// TIA Portal V20 export
FUNCTION_BLOCK "Tippler"   // FB400, LAD
{ S7_Optimized_Access := 'TRUE' }
// stored: AutoNumber false, MemoryReserve 100, SetENOAutomatically false
   VAR_INPUT
      Pallet_On_Tippler : Bool;
      iA1LowClamp_BasePos : Bool;
      iA1UpClamp_BasePos : Bool;
      iA2LowClamp_BasePos : Bool;
      iA2UpClamp_BasePos : Bool;
      iA1LowClamp_WorkPos : Bool;
      iA1UpClamp_WorkPos : Bool;
      iA2LowClamp_WorkPos : Bool;
      iA2UpClamp_WorkPos : Bool;
      iArm1_AngleValue : Int;
      iArm2_AngleValue : Int;
      iArm1_BasePos : Bool;
      iArm2_BasePos : Bool;
      HMI_Control : Bool;
      HMI_ButtonUp : Bool;
      HMI_ButtonDown : Bool;
      iButton_Down : Bool;
      iButton_Up : Bool;
   END_VAR
   VAR_OUTPUT
      Fq_Main_Valve_Arms : Bool;
      Fq_Main_Valve_Clamps : Bool;
      Fq_HydraulicUnit : Bool;
      qArm1 : Int;
      qArm2 : Int;
      qLowerClamps_Backward : Bool;
      qUpperClamps_Backward : Bool;
      qLowerClamps_Forward : Bool;
      qUpperClamps_Forward : Bool;
   END_VAR
   VAR
      Hydraulic_Ready { S7_SetPoint := 'True'} : TON_TIME;
      Hydraulic_Off { S7_SetPoint := 'True'} : TON_TIME;
      LowerClamps { S7_SetPoint := 'True'} : "Clamp";
      UpperClamps { S7_SetPoint := 'True'} : "Clamp";
      Arms { S7_SetPoint := 'True'} : "Arms";
      "Step" { S7_SetPoint := 'True'} : Int;
      ReqArmsDown : Bool;
      ReqArmsUp : Bool;
      Arms_workPos : Bool;
      Arms_basePos : Bool;
      Arms_clampsOperPos { S7_SetPoint := 'True'} : Bool;
      Tippler_maintenance { S7_SetPoint := 'True'} : "Tippler_maintenance";
      ButtonArmsDown { S7_SetPoint := 'True'} : Bool;
      ButtonArmsUp { S7_SetPoint := 'True'} : Bool;
      ReqLowerClampsClose : Bool;
      ReqUpperClampsClose : Bool;
      ReqLowerClampsOpen : Bool;
      ReqUpperClampsOpen : Bool;
      Timer_ClampsWorkPos { S7_SetPoint := 'True'} : TON_TIME;
      Timer_ClampsBasePos { S7_SetPoint := 'True'} : TON_TIME;
      Tippler_keep_down { S7_SetPoint := 'True'} : TP_TIME;
      N_Trig_Button_Down { S7_SetPoint := 'True'} : Bool;
   END_VAR
   VAR_TEMP
      Arm_Valves_Not_Actuated : Bool;
      Clamp_Valves_Not_Actuated : Bool;
   END_VAR
   VAR_TEMP   // added for the SCL form of the ladder/FBD networks
      _w1 : Bool;
   END_VAR
BEGIN

REGION Network 1: Zawory na ramionach niewysterowane
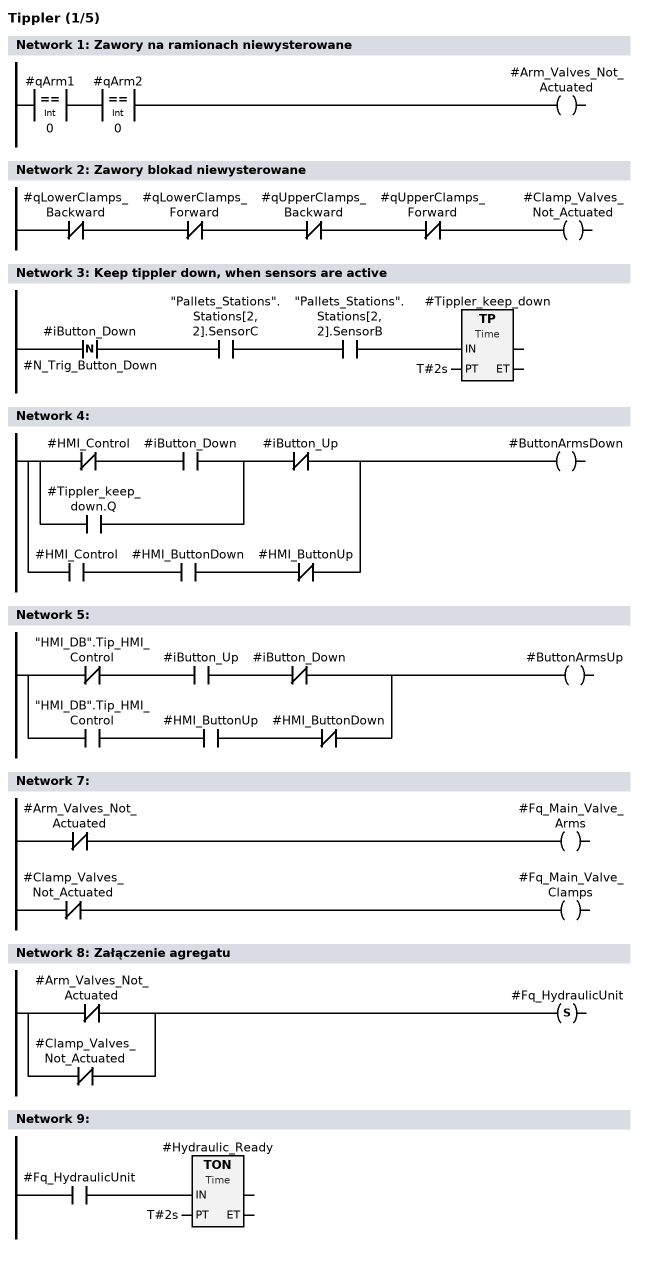
   RUNG wire#powerrail
      { S7_Templates := "SrcType := Int" } EQ_Contact(in1 := #qArm1, in2 := 0)
      { S7_Templates := "SrcType := Int" } EQ_Contact(in1 := #qArm2, in2 := 0)
      Coil( #Arm_Valves_Not_Actuated )
   END_RUNG
   // the same network as SCL:
   #Arm_Valves_Not_Actuated := (#qArm1 = 0) AND (#qArm2 = 0);
END_REGION

REGION Network 2: Zawory blokad niewysterowane
   RUNG wire#powerrail
      I_Contact( #qLowerClamps_Backward )
      I_Contact( #qLowerClamps_Forward )
      I_Contact( #qUpperClamps_Backward )
      I_Contact( #qUpperClamps_Forward )
      Coil( #Clamp_Valves_Not_Actuated )
   END_RUNG
   // the same network as SCL:
   #Clamp_Valves_Not_Actuated := NOT #qLowerClamps_Backward AND NOT #qLowerClamps_Forward AND NOT #qUpperClamps_Backward AND NOT #qUpperClamps_Forward;
END_REGION

REGION Network 3: Keep tippler down, when sensors are active
   RUNG wire#powerrail
      N_Contact(operand := #iButton_Down, bit := #N_Trig_Button_Down)
      Contact( "Pallets_Stations".Stations[2, 2].SensorC )
      Contact( "Pallets_Stations".Stations[2, 2].SensorB )
      { S7_Templates := "time_type := Time" } #Tippler_keep_down.TP(pt := T#2s, et =>)
   END_RUNG
   // the same network as SCL:
   #_w1 := NOT #iButton_Down AND #N_Trig_Button_Down;   // falling edge of #iButton_Down
   #N_Trig_Button_Down := #iButton_Down;
   #Tippler_keep_down(IN := #_w1 AND "Pallets_Stations".Stations[2, 2].SensorC AND "Pallets_Stations".Stations[2, 2].SensorB,   // TP
                      PT := T#2s);
END_REGION

REGION Network 4
   RUNG wire#powerrail
      I_Contact( #HMI_Control )
      Contact( #iButton_Down )
      wire#w1
      I_Contact( #iButton_Up )
      wire#w2
      Coil( #ButtonArmsDown )
   END_RUNG
   RUNG wire#powerrail
      Contact( #Tippler_keep_down.Q )
   END_RUNG wire#w1
   RUNG wire#powerrail
      Contact( #HMI_Control )
      Contact( #HMI_ButtonDown )
      I_Contact( #HMI_ButtonUp )
   END_RUNG wire#w2
   // the same network as SCL:
   #ButtonArmsDown := (((NOT #HMI_Control AND #iButton_Down) OR #Tippler_keep_down.Q) AND NOT #iButton_Up) OR (#HMI_Control AND #HMI_ButtonDown AND NOT #HMI_ButtonUp);
END_REGION

REGION Network 5
   RUNG wire#powerrail
      I_Contact( "HMI_DB".Tip_HMI_Control )
      Contact( #iButton_Up )
      I_Contact( #iButton_Down )
      wire#w1
      Coil( #ButtonArmsUp )
   END_RUNG
   RUNG wire#powerrail
      Contact( "HMI_DB".Tip_HMI_Control )
      Contact( #HMI_ButtonUp )
      I_Contact( #HMI_ButtonDown )
   END_RUNG wire#w1
   // the same network as SCL:
   #ButtonArmsUp := (NOT "HMI_DB".Tip_HMI_Control AND #iButton_Up AND NOT #iButton_Down) OR ("HMI_DB".Tip_HMI_Control AND #HMI_ButtonUp AND NOT #HMI_ButtonDown);
END_REGION

REGION Network 6 (SCL)
   #ReqArmsDown := 0;
   #ReqArmsUp := 0;
   #ReqLowerClampsClose := 0;
   #ReqUpperClampsClose := 0;
   #ReqLowerClampsOpen := 0;
   #ReqUpperClampsOpen := 0;
   IF "HMI_DB".Tip_MT_Control = 1 THEN
       #Step := 0;
   END_IF;
   CASE #Step OF
       0:
           IF #ButtonArmsDown THEN
               IF #Arms_basePos = 0 AND #iA1LowClamp_BasePos AND #iA2LowClamp_BasePos AND #iA1UpClamp_BasePos AND #iA2UpClamp_BasePos THEN
                   #ReqArmsDown := 1;
               ELSIF #Arms_basePos = 0 AND #Arms_clampsOperPos = 0 AND (#Arms.Arm1AngleValue > 3 OR  #Arms.Arm2AngleValue > 3) THEN
                   #ReqArmsDown := 1;
               ELSIF #Arms_clampsOperPos OR #Arms_basePos OR #Pallet_On_Tippler = 0 THEN
                   IF #iA1LowClamp_BasePos = 0 OR #iA2LowClamp_BasePos = 0 THEN
                       #ReqLowerClampsOpen := 1;
                   END_IF;
                   IF #iA1UpClamp_BasePos = 0 OR #iA2UpClamp_BasePos = 0 THEN
                       #ReqUpperClampsOpen := 1;
                   END_IF;
               END_IF;
               IF  #iA1LowClamp_BasePos AND #iA1UpClamp_BasePos AND #iA2LowClamp_BasePos AND #iA2UpClamp_BasePos THEN
                   #Step += 1;
               END_IF;
           END_IF;

           1:
               IF #ButtonArmsUp AND NOT #Arms_clampsOperPos AND #Arms.Arm1AngleValue < 4 AND #Arms.Arm2AngleValue < 4 THEN
                   #ReqArmsUp := 1;
               ELSIF #ButtonArmsDown AND #Arms_basePos = 0 THEN
                   #ReqArmsDown := 1;
               ELSIF #ButtonArmsUp AND #Arms_clampsOperPos THEN
                   //#ReqArmsUp := 0;
                   #Step += 1;
               END_IF;

       2:
           IF #ButtonArmsUp AND #Arms.Arm1AngleValue < 12 AND #Arms.Arm2AngleValue < 12 THEN
               IF NOT #Timer_ClampsWorkPos.Q THEN
                   #ReqUpperClampsClose := 1;
                   #ReqLowerClampsClose := 1;
                   #ReqArmsUp := 1;
               END_IF;
           ELSIF #ButtonArmsDown THEN
               IF #Timer_ClampsBasePos.Q = 0 THEN
                   #ReqLowerClampsOpen := 1;
                   #ReqUpperClampsOpen := 1;
               END_IF;
           END_IF;
           #Timer_ClampsWorkPos(IN:= #Step = 2 AND #ButtonArmsUp AND #iA1LowClamp_WorkPos AND #iA1UpClamp_WorkPos AND #iA2LowClamp_WorkPos AND #iA2UpClamp_WorkPos,
                                PT:=t#3s);
           IF (#Timer_ClampsWorkPos.Q) THEN
               #Step += 1;
           END_IF;
           #Timer_ClampsBasePos(IN:= #Step = 2 AND #ButtonArmsDown AND #iA1LowClamp_BasePos AND #iA1UpClamp_BasePos AND #iA2LowClamp_BasePos AND #iA2UpClamp_BasePos ,
                                PT:=t#3s);

           IF #Timer_ClampsBasePos.Q THEN
               #Step -= 1;
           END_IF;
       3:
           IF #ButtonArmsUp AND #Arms_workPos = 0 AND #iA1LowClamp_WorkPos AND #iA1UpClamp_WorkPos AND #iA2LowClamp_WorkPos AND #iA2UpClamp_WorkPos THEN
               #ReqArmsUp := 1;
           ELSIF #ButtonArmsDown AND #Arms_clampsOperPos = 0 AND #iA1LowClamp_WorkPos AND #iA1UpClamp_WorkPos AND #iA2LowClamp_WorkPos AND #iA2UpClamp_WorkPos THEN
               #ReqArmsDown := 1;
           ELSIF #ButtonArmsUp AND #Arms_workPos = 1 AND #iA1LowClamp_WorkPos AND #iA1UpClamp_WorkPos AND #iA2LowClamp_WorkPos AND #iA2UpClamp_WorkPos THEN
               #Step := 4;
           ELSIF #ButtonArmsDown AND #Arms_clampsOperPos THEN
               #ReqArmsDown := 0;
               #Step := 2;
           END_IF;
       4:
           IF #ButtonArmsDown AND #Arms_clampsOperPos = 0 AND #iA1LowClamp_WorkPos AND #iA1UpClamp_WorkPos AND #iA2LowClamp_WorkPos AND #iA2UpClamp_WorkPos THEN
               #Step := 3;
           END_IF;
       ELSE
           #Step := 0;
   END_CASE;
END_REGION

REGION Network 7
   RUNG wire#powerrail
      I_Contact( #Arm_Valves_Not_Actuated )
      Coil( #Fq_Main_Valve_Arms )
   END_RUNG
   RUNG wire#powerrail
      I_Contact( #Clamp_Valves_Not_Actuated )
      Coil( #Fq_Main_Valve_Clamps )
   END_RUNG
   // the same network as SCL:
   #Fq_Main_Valve_Arms := NOT #Arm_Valves_Not_Actuated;
   #Fq_Main_Valve_Clamps := NOT #Clamp_Valves_Not_Actuated;
END_REGION

REGION Network 8: Załączenie agregatu
   RUNG wire#powerrail
      I_Contact( #Arm_Valves_Not_Actuated )
      wire#w1
      S_Coil( #Fq_HydraulicUnit )
   END_RUNG
   RUNG wire#powerrail
      I_Contact( #Clamp_Valves_Not_Actuated )
   END_RUNG wire#w1
   // the same network as SCL:
   IF NOT #Arm_Valves_Not_Actuated OR NOT #Clamp_Valves_Not_Actuated THEN #Fq_HydraulicUnit := TRUE; END_IF;
END_REGION

REGION Network 9
   RUNG wire#powerrail
      Contact( #Fq_HydraulicUnit )
      { S7_Templates := "time_type := Time" } #Hydraulic_Ready.TON(pt := T#2s, et =>)
   END_RUNG
   // the same network as SCL:
   #Hydraulic_Ready(IN := #Fq_HydraulicUnit, PT := T#2s);   // TON
END_REGION

REGION Network 10: Czasowe wyłączenie po braku działania
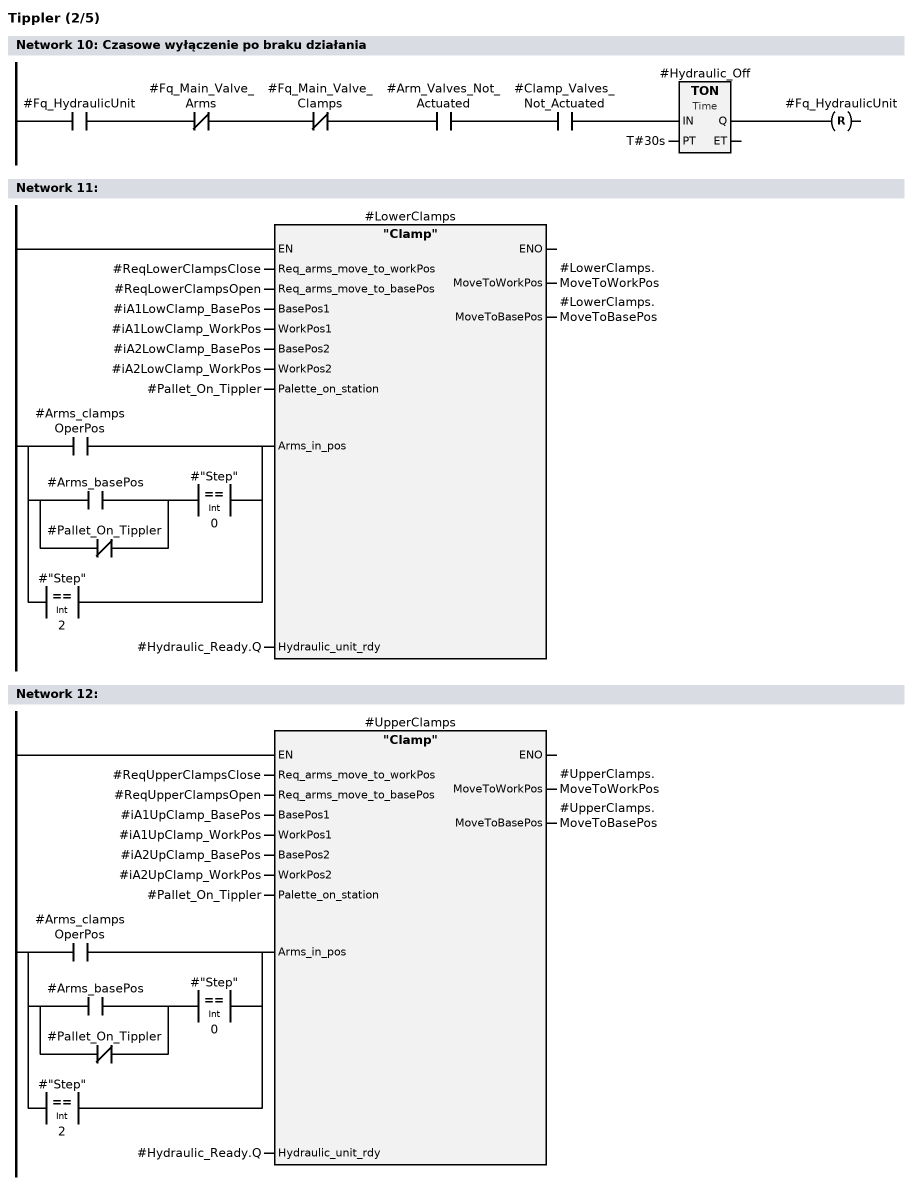
   RUNG wire#powerrail
      Contact( #Fq_HydraulicUnit )
      I_Contact( #Fq_Main_Valve_Arms )
      I_Contact( #Fq_Main_Valve_Clamps )
      Contact( #Arm_Valves_Not_Actuated )
      Contact( #Clamp_Valves_Not_Actuated )
      { S7_Templates := "time_type := Time" } #Hydraulic_Off.TON(pt := T#30s, et =>)
      R_Coil( #Fq_HydraulicUnit )
   END_RUNG
   // the same network as SCL:
   #Hydraulic_Off(IN := #Fq_HydraulicUnit AND NOT #Fq_Main_Valve_Arms AND NOT #Fq_Main_Valve_Clamps AND #Arm_Valves_Not_Actuated AND #Clamp_Valves_Not_Actuated,   // TON
                  PT := T#30s);
   IF #Hydraulic_Off.Q THEN #Fq_HydraulicUnit := FALSE; END_IF;
END_REGION

REGION Network 11
   RUNG wire#powerrail
      #LowerClamps(Arms_in_pos := wire#w2, Req_arms_move_to_workPos := #ReqLowerClampsClose, Req_arms_move_to_basePos := #ReqLowerClampsOpen, BasePos1 := #iA1LowClamp_BasePos, WorkPos1 := #iA1LowClamp_WorkPos, BasePos2 := #iA2LowClamp_BasePos, WorkPos2 := #iA2LowClamp_WorkPos, Palette_on_station := #Pallet_On_Tippler, Hydraulic_unit_rdy := #Hydraulic_Ready.Q, MoveToWorkPos => #LowerClamps.MoveToWorkPos, MoveToBasePos => #LowerClamps.MoveToBasePos)
   END_RUNG
   RUNG wire#powerrail
      Contact( #Arms_clampsOperPos )
   END_RUNG wire#w2
   RUNG wire#powerrail
      Contact( #Arms_basePos )
      wire#w1
      { S7_Templates := "SrcType := Int" } EQ_Contact(in1 := #"Step", in2 := 0)
   END_RUNG wire#w2
   RUNG wire#powerrail
      I_Contact( #Pallet_On_Tippler )
   END_RUNG wire#w1
   RUNG wire#powerrail
      { S7_Templates := "SrcType := Int" } EQ_Contact(in1 := #"Step", in2 := 2)
   END_RUNG wire#w2
   // the same network as SCL:
   #LowerClamps(Req_arms_move_to_workPos := #ReqLowerClampsClose,   // "Clamp"
                Req_arms_move_to_basePos := #ReqLowerClampsOpen,
                BasePos1 := #iA1LowClamp_BasePos,
                WorkPos1 := #iA1LowClamp_WorkPos,
                BasePos2 := #iA2LowClamp_BasePos,
                WorkPos2 := #iA2LowClamp_WorkPos,
                Palette_on_station := #Pallet_On_Tippler,
                Arms_in_pos := #Arms_clampsOperPos OR ((#Arms_basePos OR NOT #Pallet_On_Tippler) AND (#"Step" = 0)) OR (#"Step" = 2),
                Hydraulic_unit_rdy := #Hydraulic_Ready.Q,
                MoveToWorkPos => #LowerClamps.MoveToWorkPos,
                MoveToBasePos => #LowerClamps.MoveToBasePos);
END_REGION

REGION Network 12
   RUNG wire#powerrail
      #UpperClamps(Arms_in_pos := wire#w2, Req_arms_move_to_workPos := #ReqUpperClampsClose, Req_arms_move_to_basePos := #ReqUpperClampsOpen, BasePos1 := #iA1UpClamp_BasePos, WorkPos1 := #iA1UpClamp_WorkPos, BasePos2 := #iA2UpClamp_BasePos, WorkPos2 := #iA2UpClamp_WorkPos, Palette_on_station := #Pallet_On_Tippler, Hydraulic_unit_rdy := #Hydraulic_Ready.Q, MoveToWorkPos => #UpperClamps.MoveToWorkPos, MoveToBasePos => #UpperClamps.MoveToBasePos)
   END_RUNG
   RUNG wire#powerrail
      Contact( #Arms_clampsOperPos )
   END_RUNG wire#w2
   RUNG wire#powerrail
      Contact( #Arms_basePos )
      wire#w1
      { S7_Templates := "SrcType := Int" } EQ_Contact(in1 := #"Step", in2 := 0)
   END_RUNG wire#w2
   RUNG wire#powerrail
      I_Contact( #Pallet_On_Tippler )
   END_RUNG wire#w1
   RUNG wire#powerrail
      { S7_Templates := "SrcType := Int" } EQ_Contact(in1 := #"Step", in2 := 2)
   END_RUNG wire#w2
   // the same network as SCL:
   #UpperClamps(Req_arms_move_to_workPos := #ReqUpperClampsClose,   // "Clamp"
                Req_arms_move_to_basePos := #ReqUpperClampsOpen,
                BasePos1 := #iA1UpClamp_BasePos,
                WorkPos1 := #iA1UpClamp_WorkPos,
                BasePos2 := #iA2UpClamp_BasePos,
                WorkPos2 := #iA2UpClamp_WorkPos,
                Palette_on_station := #Pallet_On_Tippler,
                Arms_in_pos := #Arms_clampsOperPos OR ((#Arms_basePos OR NOT #Pallet_On_Tippler) AND (#"Step" = 0)) OR (#"Step" = 2),
                Hydraulic_unit_rdy := #Hydraulic_Ready.Q,
                MoveToWorkPos => #UpperClamps.MoveToWorkPos,
                MoveToBasePos => #UpperClamps.MoveToBasePos);
END_REGION

REGION Network 13
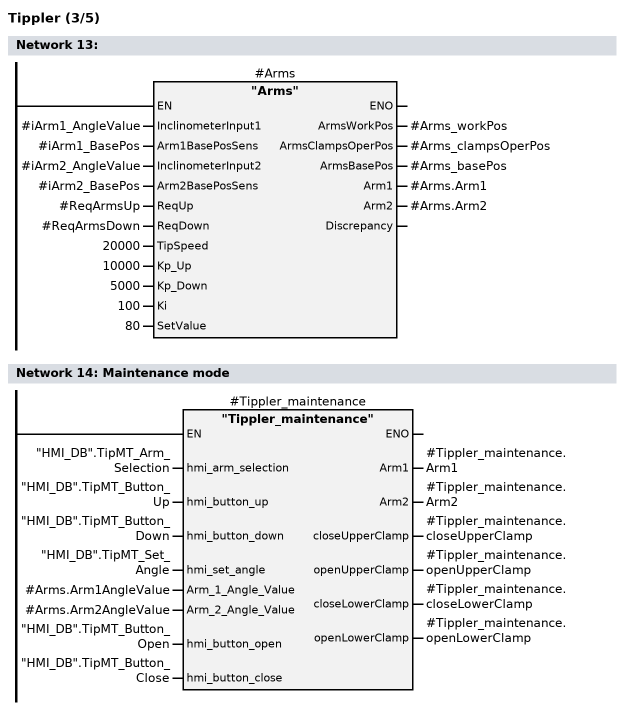
   RUNG wire#powerrail
      #Arms(InclinometerInput1 := #iArm1_AngleValue, Arm1BasePosSens := #iArm1_BasePos, InclinometerInput2 := #iArm2_AngleValue, Arm2BasePosSens := #iArm2_BasePos, ReqUp := #ReqArmsUp, ReqDown := #ReqArmsDown, TipSpeed := 20000, Kp_Up := 10000, Kp_Down := 5000, Ki := 100, SetValue := 80, ArmsWorkPos => #Arms_workPos, ArmsClampsOperPos => #Arms_clampsOperPos, ArmsBasePos => #Arms_basePos, Arm1 => #Arms.Arm1, Arm2 => #Arms.Arm2, Discrepancy =>)
   END_RUNG
   // the same network as SCL:
   #Arms(InclinometerInput1 := #iArm1_AngleValue,   // "Arms"
         Arm1BasePosSens := #iArm1_BasePos,
         InclinometerInput2 := #iArm2_AngleValue,
         Arm2BasePosSens := #iArm2_BasePos,
         ReqUp := #ReqArmsUp,
         ReqDown := #ReqArmsDown,
         TipSpeed := 20000,
         Kp_Up := 10000,
         Kp_Down := 5000,
         Ki := 100,
         SetValue := 80,
         ArmsWorkPos => #Arms_workPos,
         ArmsClampsOperPos => #Arms_clampsOperPos,
         ArmsBasePos => #Arms_basePos,
         Arm1 => #Arms.Arm1,
         Arm2 => #Arms.Arm2);
END_REGION

REGION Network 14: Maintenance mode
   RUNG wire#powerrail
      #Tippler_maintenance(hmi_arm_selection := "HMI_DB".TipMT_Arm_Selection, hmi_button_up := "HMI_DB".TipMT_Button_Up, hmi_button_down := "HMI_DB".TipMT_Button_Down, hmi_set_angle := "HMI_DB".TipMT_Set_Angle, Arm_1_Angle_Value := #Arms.Arm1AngleValue, Arm_2_Angle_Value := #Arms.Arm2AngleValue, hmi_button_open := "HMI_DB".TipMT_Button_Open, hmi_button_close := "HMI_DB".TipMT_Button_Close, Arm1 => #Tippler_maintenance.Arm1, Arm2 => #Tippler_maintenance.Arm2, closeUpperClamp => #Tippler_maintenance.closeUpperClamp, openUpperClamp => #Tippler_maintenance.openUpperClamp, closeLowerClamp => #Tippler_maintenance.closeLowerClamp, openLowerClamp => #Tippler_maintenance.openLowerClamp)
   END_RUNG
   // the same network as SCL:
   #Tippler_maintenance(hmi_arm_selection := "HMI_DB".TipMT_Arm_Selection,   // "Tippler_maintenance"
                        hmi_button_up := "HMI_DB".TipMT_Button_Up,
                        hmi_button_down := "HMI_DB".TipMT_Button_Down,
                        hmi_set_angle := "HMI_DB".TipMT_Set_Angle,
                        Arm_1_Angle_Value := #Arms.Arm1AngleValue,
                        Arm_2_Angle_Value := #Arms.Arm2AngleValue,
                        hmi_button_open := "HMI_DB".TipMT_Button_Open,
                        hmi_button_close := "HMI_DB".TipMT_Button_Close,
                        Arm1 => #Tippler_maintenance.Arm1,
                        Arm2 => #Tippler_maintenance.Arm2,
                        closeUpperClamp => #Tippler_maintenance.closeUpperClamp,
                        openUpperClamp => #Tippler_maintenance.openUpperClamp,
                        closeLowerClamp => #Tippler_maintenance.closeLowerClamp,
                        openLowerClamp => #Tippler_maintenance.openLowerClamp);
END_REGION

REGION Network 15: Arm Valves Control
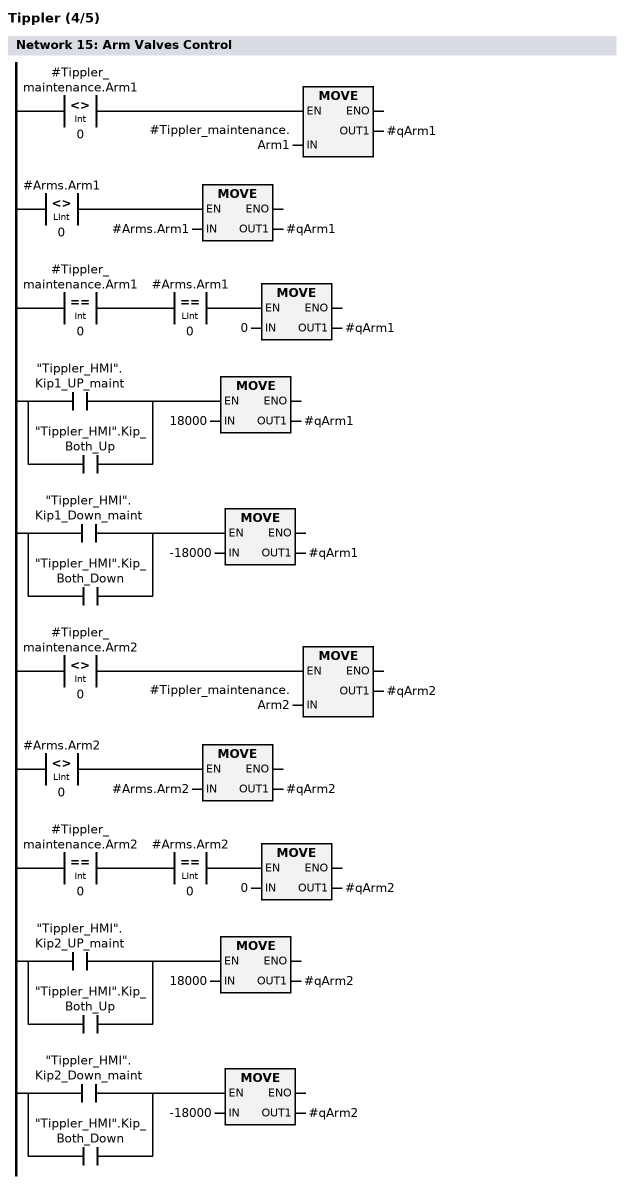
   RUNG wire#powerrail
      { S7_Templates := "SrcType := Int" } NE_Contact(in1 := #Tippler_maintenance.Arm1, in2 := 0)
      Move(in := #Tippler_maintenance.Arm1, out1 => #qArm1)
   END_RUNG
   RUNG wire#powerrail
      { S7_Templates := "SrcType := LInt" } NE_Contact(in1 := #Arms.Arm1, in2 := 0)
      Move(in := #Arms.Arm1, out1 => #qArm1)
   END_RUNG
   RUNG wire#powerrail
      { S7_Templates := "SrcType := Int" } EQ_Contact(in1 := #Tippler_maintenance.Arm1, in2 := 0)
      { S7_Templates := "SrcType := LInt" } EQ_Contact(in1 := #Arms.Arm1, in2 := 0)
      Move(in := 0, out1 => #qArm1)
   END_RUNG
   RUNG wire#powerrail
      Contact( "Tippler_HMI".Kip1_UP_maint )
      wire#w1
      Move(in := 18000, out1 => #qArm1)
   END_RUNG
   RUNG wire#powerrail
      Contact( "Tippler_HMI".Kip_Both_Up )
   END_RUNG wire#w1
   RUNG wire#powerrail
      Contact( "Tippler_HMI".Kip1_Down_maint )
      wire#w2
      Move(in := -18000, out1 => #qArm1)
   END_RUNG
   RUNG wire#powerrail
      Contact( "Tippler_HMI".Kip_Both_Down )
   END_RUNG wire#w2
   RUNG wire#powerrail
      { S7_Templates := "SrcType := Int" } NE_Contact(in1 := #Tippler_maintenance.Arm2, in2 := 0)
      Move(in := #Tippler_maintenance.Arm2, out1 => #qArm2)
   END_RUNG
   RUNG wire#powerrail
      { S7_Templates := "SrcType := LInt" } NE_Contact(in1 := #Arms.Arm2, in2 := 0)
      Move(in := #Arms.Arm2, out1 => #qArm2)
   END_RUNG
   RUNG wire#powerrail
      { S7_Templates := "SrcType := Int" } EQ_Contact(in1 := #Tippler_maintenance.Arm2, in2 := 0)
      { S7_Templates := "SrcType := LInt" } EQ_Contact(in1 := #Arms.Arm2, in2 := 0)
      Move(in := 0, out1 => #qArm2)
   END_RUNG
   RUNG wire#powerrail
      Contact( "Tippler_HMI".Kip2_UP_maint )
      wire#w3
      Move(in := 18000, out1 => #qArm2)
   END_RUNG
   RUNG wire#powerrail
      Contact( "Tippler_HMI".Kip_Both_Up )
   END_RUNG wire#w3
   RUNG wire#powerrail
      Contact( "Tippler_HMI".Kip2_Down_maint )
      wire#w4
      Move(in := -18000, out1 => #qArm2)
   END_RUNG
   RUNG wire#powerrail
      Contact( "Tippler_HMI".Kip_Both_Down )
   END_RUNG wire#w4
   // the same network as SCL:
   IF #Tippler_maintenance.Arm1 <> 0 THEN #qArm1 := #Tippler_maintenance.Arm1; END_IF;
   IF #Arms.Arm1 <> 0 THEN #qArm1 := #Arms.Arm1; END_IF;
   IF (#Tippler_maintenance.Arm1 = 0) AND (#Arms.Arm1 = 0) THEN #qArm1 := 0; END_IF;
   IF "Tippler_HMI".Kip1_UP_maint OR "Tippler_HMI".Kip_Both_Up THEN #qArm1 := 18000; END_IF;
   IF "Tippler_HMI".Kip1_Down_maint OR "Tippler_HMI".Kip_Both_Down THEN #qArm1 := -18000; END_IF;
   IF #Tippler_maintenance.Arm2 <> 0 THEN #qArm2 := #Tippler_maintenance.Arm2; END_IF;
   IF #Arms.Arm2 <> 0 THEN #qArm2 := #Arms.Arm2; END_IF;
   IF (#Tippler_maintenance.Arm2 = 0) AND (#Arms.Arm2 = 0) THEN #qArm2 := 0; END_IF;
   IF "Tippler_HMI".Kip2_UP_maint OR "Tippler_HMI".Kip_Both_Up THEN #qArm2 := 18000; END_IF;
   IF "Tippler_HMI".Kip2_Down_maint OR "Tippler_HMI".Kip_Both_Down THEN #qArm2 := -18000; END_IF;
END_REGION

REGION Network 16: Clamps Valve Control
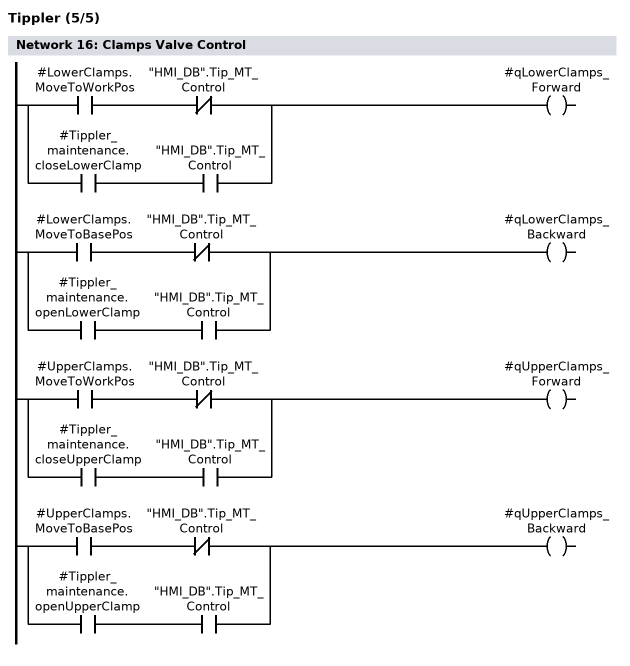
   RUNG wire#powerrail
      Contact( #LowerClamps.MoveToWorkPos )
      I_Contact( "HMI_DB".Tip_MT_Control )
      wire#w1
      Coil( #qLowerClamps_Forward )
   END_RUNG
   RUNG wire#powerrail
      Contact( #Tippler_maintenance.closeLowerClamp )
      Contact( "HMI_DB".Tip_MT_Control )
   END_RUNG wire#w1
   RUNG wire#powerrail
      Contact( #LowerClamps.MoveToBasePos )
      I_Contact( "HMI_DB".Tip_MT_Control )
      wire#w2
      Coil( #qLowerClamps_Backward )
   END_RUNG
   RUNG wire#powerrail
      Contact( #Tippler_maintenance.openLowerClamp )
      Contact( "HMI_DB".Tip_MT_Control )
   END_RUNG wire#w2
   RUNG wire#powerrail
      Contact( #UpperClamps.MoveToWorkPos )
      I_Contact( "HMI_DB".Tip_MT_Control )
      wire#w3
      Coil( #qUpperClamps_Forward )
   END_RUNG
   RUNG wire#powerrail
      Contact( #Tippler_maintenance.closeUpperClamp )
      Contact( "HMI_DB".Tip_MT_Control )
   END_RUNG wire#w3
   RUNG wire#powerrail
      Contact( #UpperClamps.MoveToBasePos )
      I_Contact( "HMI_DB".Tip_MT_Control )
      wire#w4
      Coil( #qUpperClamps_Backward )
   END_RUNG
   RUNG wire#powerrail
      Contact( #Tippler_maintenance.openUpperClamp )
      Contact( "HMI_DB".Tip_MT_Control )
   END_RUNG wire#w4
   // the same network as SCL:
   #qLowerClamps_Forward := (#LowerClamps.MoveToWorkPos AND NOT "HMI_DB".Tip_MT_Control) OR (#Tippler_maintenance.closeLowerClamp AND "HMI_DB".Tip_MT_Control);
   #qLowerClamps_Backward := (#LowerClamps.MoveToBasePos AND NOT "HMI_DB".Tip_MT_Control) OR (#Tippler_maintenance.openLowerClamp AND "HMI_DB".Tip_MT_Control);
   #qUpperClamps_Forward := (#UpperClamps.MoveToWorkPos AND NOT "HMI_DB".Tip_MT_Control) OR (#Tippler_maintenance.closeUpperClamp AND "HMI_DB".Tip_MT_Control);
   #qUpperClamps_Backward := (#UpperClamps.MoveToBasePos AND NOT "HMI_DB".Tip_MT_Control) OR (#Tippler_maintenance.openUpperClamp AND "HMI_DB".Tip_MT_Control);
END_REGION
END_FUNCTION_BLOCK
